// Mitsubishi GX Works2 project: 파이썬   PLC: Q03UDV

PROGRAM MAIN
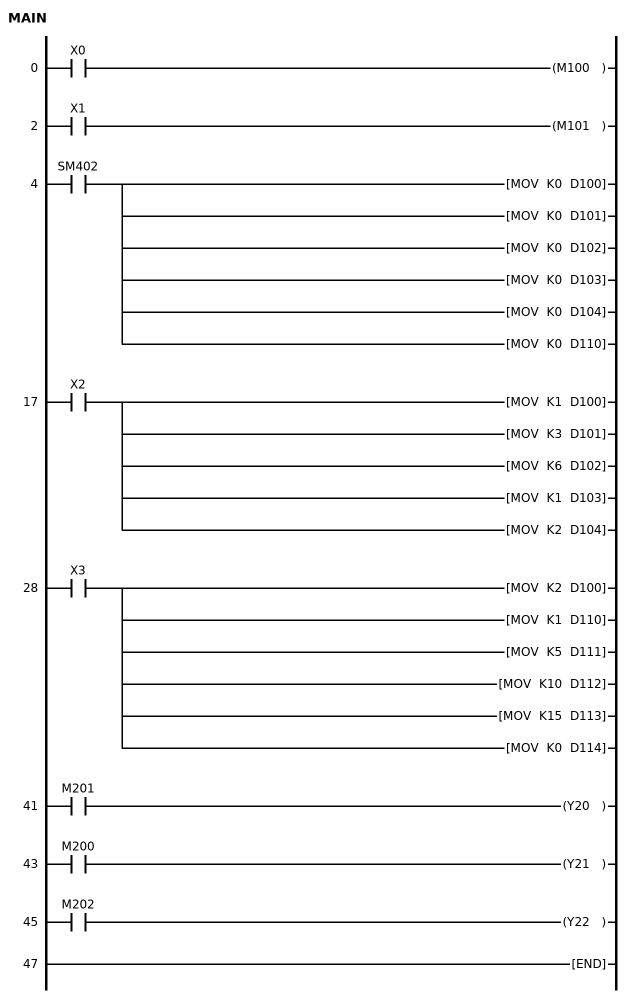
0     LD      X0
      OUT     M100
2     LD      X1
      OUT     M101
4     LD      SM402
      MOV     K0 D100
      MOV     K0 D101
      MOV     K0 D102
      MOV     K0 D103
      MOV     K0 D104
      MOV     K0 D110
17    LD      X2
      MOV     K1 D100
      MOV     K3 D101
      MOV     K6 D102
      MOV     K1 D103
      MOV     K2 D104
28    LD      X3
      MOV     K2 D100
      MOV     K1 D110
      MOV     K5 D111
      MOV     K10 D112
      MOV     K15 D113
      MOV     K0 D114
41    LD      M201
      OUT     Y20
43    LD      M200
      OUT     Y21
45    LD      M202
      OUT     Y22
47    END
END_PROGRAM
